% RSLogix 500 project I2P JOB 27 - SOLUTION_BAK003.RSS, saved by version 10.00.00.00 %
PROJECT "UNTITLED"    % processor: Bul.1763 MicroLogix 1100 Series B %

PROGRAM FILES
  LAD 2   12 rungs

DATA FILES
  O0 OUTPUT  4 elements
  I1 INPUT  6 elements
  S2 STATUS  66 elements
  B3 BINARY  3 elements
  T4 TIMER  1 elements
  C5 COUNTER  1 elements
  R6 CONTROL  1 elements
  N7 INTEGER  1 elements
  F8 FLOAT  3 elements

LADDER 2
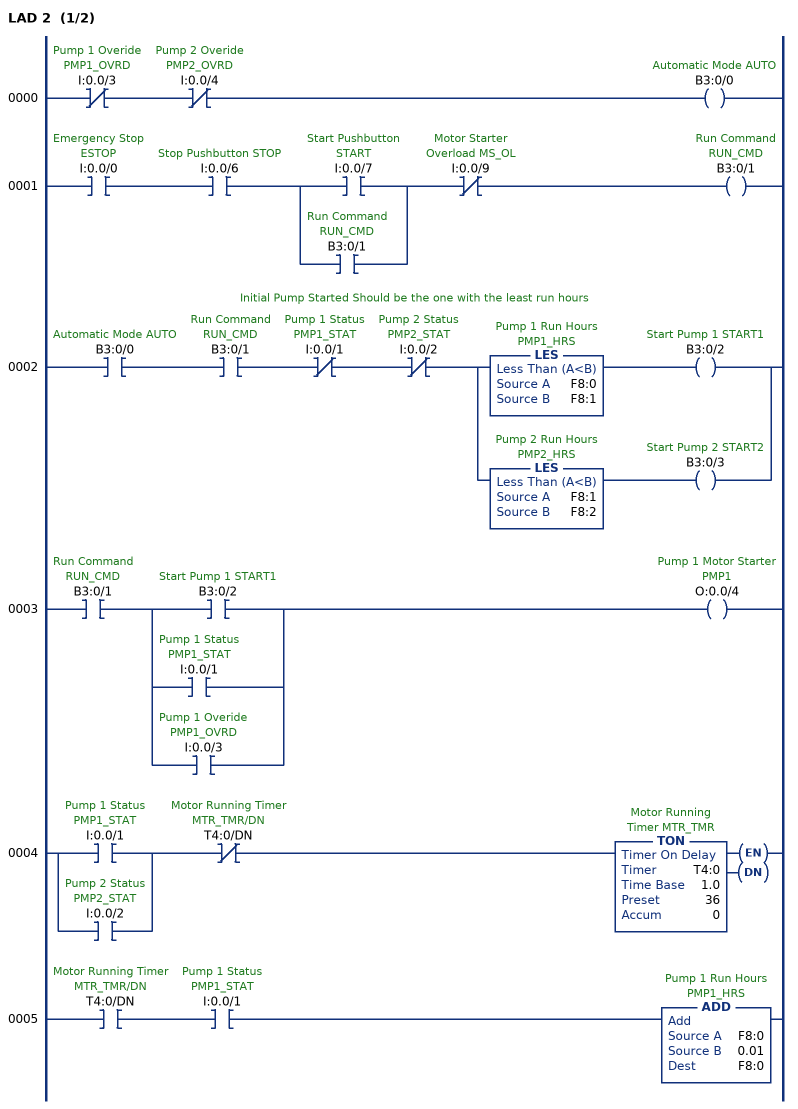
% Rung: 0 %
SOR XIO I:0.0/3 XIO I:0.0/4 OTE B3:0/0 EOR
%   I:0.0/3  PMP1_OVRD  "Pump 1 Overide" %
%   I:0.0/4  PMP2_OVRD  "Pump 2 Overide" %
%   B3:0/0  AUTO  "Automatic Mode" %
% Rung: 1 %
SOR XIC I:0.0/0 XIC I:0.0/6 BST XIC I:0.0/7 NXB XIC B3:0/1 BND XIO I:0.0/9 OTE B3:0/1 EOR
%   I:0.0/0  ESTOP  "Emergency Stop" %
%   I:0.0/6  STOP  "Stop Pushbutton" %
%   I:0.0/7  START  "Start Pushbutton" %
%   B3:0/1  RUN_CMD  "Run Command" %
%   I:0.0/9  MS_OL  "Motor Starter Overload" %
% Rung: 2 %
% Initial Pump Started Should be the one with the least run hours %
SOR XIC B3:0/0 XIC B3:0/1 XIO I:0.0/1 XIO I:0.0/2 BST LES F8:0 F8:1 OTE B3:0/2 NXB LES F8:1 F8:2 OTE B3:0/3 BND EOR
%   B3:0/0  AUTO  "Automatic Mode" %
%   B3:0/1  RUN_CMD  "Run Command" %
%   I:0.0/1  PMP1_STAT  "Pump 1 Status" %
%   I:0.0/2  PMP2_STAT  "Pump 2 Status" %
%   F8:0  PMP1_HRS  "Pump 1 Run Hours" %
%   F8:1  PMP2_HRS  "Pump 2 Run Hours" %
%   B3:0/2  START1  "Start Pump 1" %
%   F8:2  STRT_HRS  "Start Hours" %
%   B3:0/3  START2  "Start Pump 2" %
% Rung: 3 %
SOR XIC B3:0/1 BST XIC B3:0/2 NXB XIC I:0.0/1 NXB XIC I:0.0/3 BND OTE O:0.0/4 EOR
%   B3:0/1  RUN_CMD  "Run Command" %
%   B3:0/2  START1  "Start Pump 1" %
%   I:0.0/1  PMP1_STAT  "Pump 1 Status" %
%   I:0.0/3  PMP1_OVRD  "Pump 1 Overide" %
%   O:0.0/4  PMP1  "Pump 1 Motor Starter" %
% Rung: 4 %
SOR BST XIC I:0.0/1 NXB XIC I:0.0/2 BND XIO T4:0/DN TON T4:0 1.0 36 0 EOR
%   I:0.0/1  PMP1_STAT  "Pump 1 Status" %
%   I:0.0/2  PMP2_STAT  "Pump 2 Status" %
%   T4:0  MTR_TMR  "Motor Running Timer" %
% Rung: 5 %
SOR XIC T4:0/DN XIC I:0.0/1 ADD F8:0 0.01 F8:0 EOR
%   T4:0  MTR_TMR  "Motor Running Timer" %
%   I:0.0/1  PMP1_STAT  "Pump 1 Status" %
%   F8:0  PMP1_HRS  "Pump 1 Run Hours" %

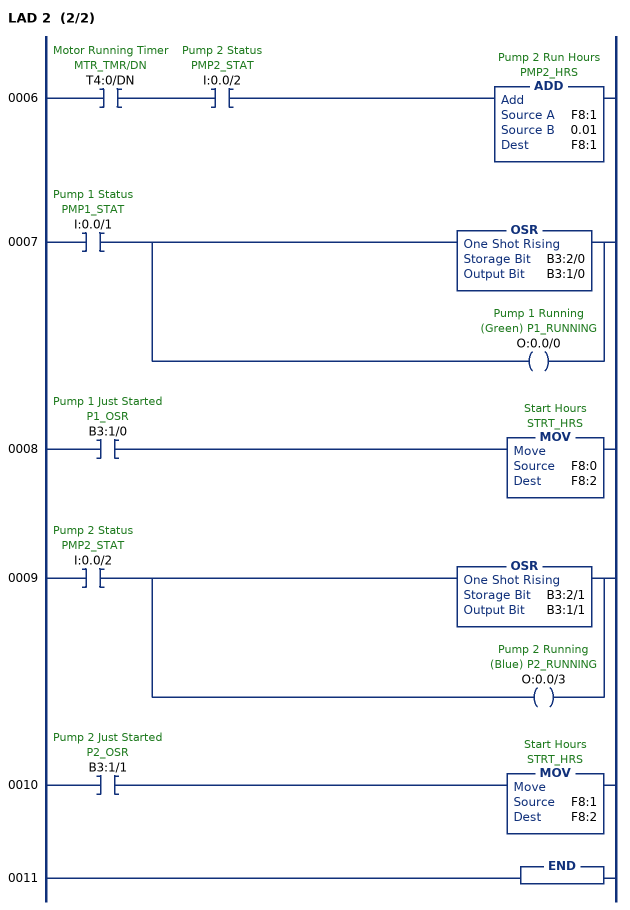
% Rung: 6 %
SOR XIC T4:0/DN XIC I:0.0/2 ADD F8:1 0.01 F8:1 EOR
%   T4:0  MTR_TMR  "Motor Running Timer" %
%   I:0.0/2  PMP2_STAT  "Pump 2 Status" %
%   F8:1  PMP2_HRS  "Pump 2 Run Hours" %
% Rung: 7 %
SOR XIC I:0.0/1 BST OSR B3:2/0 B3:1/0 NXB OTE O:0.0/0 BND EOR
%   I:0.0/1  PMP1_STAT  "Pump 1 Status" %
%   B3:1/0  P1_OSR  "Pump 1 Just Started" %
%   O:0.0/0  P1_RUNNING  "Pump 1 Running (Green)" %
% Rung: 8 %
SOR XIC B3:1/0 MOV F8:0 F8:2 EOR
%   B3:1/0  P1_OSR  "Pump 1 Just Started" %
%   F8:0  PMP1_HRS  "Pump 1 Run Hours" %
%   F8:2  STRT_HRS  "Start Hours" %
% Rung: 9 %
SOR XIC I:0.0/2 BST OSR B3:2/1 B3:1/1 NXB OTE O:0.0/3 BND EOR
%   I:0.0/2  PMP2_STAT  "Pump 2 Status" %
%   B3:1/1  P2_OSR  "Pump 2 Just Started" %
%   O:0.0/3  P2_RUNNING  "Pump 2 Running (Blue)" %
% Rung: 10 %
SOR XIC B3:1/1 MOV F8:1 F8:2 EOR
%   B3:1/1  P2_OSR  "Pump 2 Just Started" %
%   F8:1  PMP2_HRS  "Pump 2 Run Hours" %
%   F8:2  STRT_HRS  "Start Hours" %
% Rung: 11 %
SOR END EOR

DATA TABLE (non-zero values as saved)
DATA T4
% .PRE .ACC %
% T4:0 % 36 0
